// TIA Portal project "teste2" (V18)

(* hardware
DEVICE "S7-1200 station_1"  S7-1200 Station
   slot 0: "Rack_0"  S7-1200 Rack  Rack  V1.0
   slot 1: "PLC_1"  CPU 1214C AC/DC/Rly  6ES7 214-1BG40-0XB0  V4.5
   slot 2: "DI 16/DQ 16x24VDC_1"  6ES7 223-1BL32-0XB0  V2.0
   slot 3: "AI 8x13BIT_1"  6ES7 231-4HF32-0XB0  V2.1
*)

// ===== PLC "PLC_1"  CPU 1214C AC/DC/Rly =====

VAR_GLOBAL   // PLC tag table "Default tag table"
   "LED_Verde" AT %Q0.1 : Bool;
   "Bot_Emergencia" AT %I1.0 : Bool;
   "Bot_Verde" AT %I0.1 : Bool;
   "Tag_4" AT %M0.0 : Bool;
   "LED_Vermelho" AT %Q0.3 : Bool;
   "Bot_Reset" AT %I0.3 : Bool;
   "Parada" AT %M0.1 : Bool;
   "LED_Yellow" AT %Q0.2 : Bool;
   "Tag_1" AT %M0.2 : Bool;
   "Tag_2" AT %M0.3 : Bool;
   "Tag_3" AT %IW112 : Int;
   "norm" AT %MD68 : Real;
   "Angulo" AT %MW66 : Int;
   "Tag_5" AT %M0.6 : Bool;
END_VAR

TYPE "User_data_type_1"
   STRUCT
      Min_Norm : Int := 0;
      Max_Norm : Int := 27648;
   END_STRUCT;
END_TYPE

// folder: System blocks/Program resources

DATA_BLOCK "IEC_Timer_0_DB"   // DB1
{ S7_Optimized_Access := 'TRUE' }
AUTHOR : Simatic
FAMILY : IEC
NAME : IEC_TMR
VERSION : 1.0
// stored: InstanceOfName IEC_TIMER
"IEC_TIMER"
BEGIN
END_DATA_BLOCK

DATA_BLOCK "IEC_Timer_0_DB_1"   // DB2
{ S7_Optimized_Access := 'TRUE' }
AUTHOR : Simatic
FAMILY : IEC
NAME : IEC_TMR
VERSION : 1.0
// stored: InstanceOfName IEC_TIMER
"IEC_TIMER"
BEGIN
END_DATA_BLOCK

DATA_BLOCK "IEC_Timer_0_DB_2"   // DB3
{ S7_Optimized_Access := 'TRUE' }
AUTHOR : Simatic
FAMILY : IEC
NAME : IEC_TMR
VERSION : 1.0
// stored: InstanceOfName IEC_TIMER
"IEC_TIMER"
BEGIN
END_DATA_BLOCK

// folder: (top level)

ORGANIZATION_BLOCK "Main"   // OB1, LAD, ProgramCycle
TITLE = "Main Program Sweep (Cycle)"
{ S7_Optimized_Access := 'TRUE' }
VERSION : 0.1
   VAR_INPUT
      Initial_Call : Bool;   // Initial call of this OB
      Remanence : Bool;   // =True, if remanent data are available
   END_VAR
   VAR_TEMP   // added for the SCL form of the ladder/FBD networks
      _w1 : Bool;
      _w2 : Bool;
   END_VAR
BEGIN

REGION Network 1
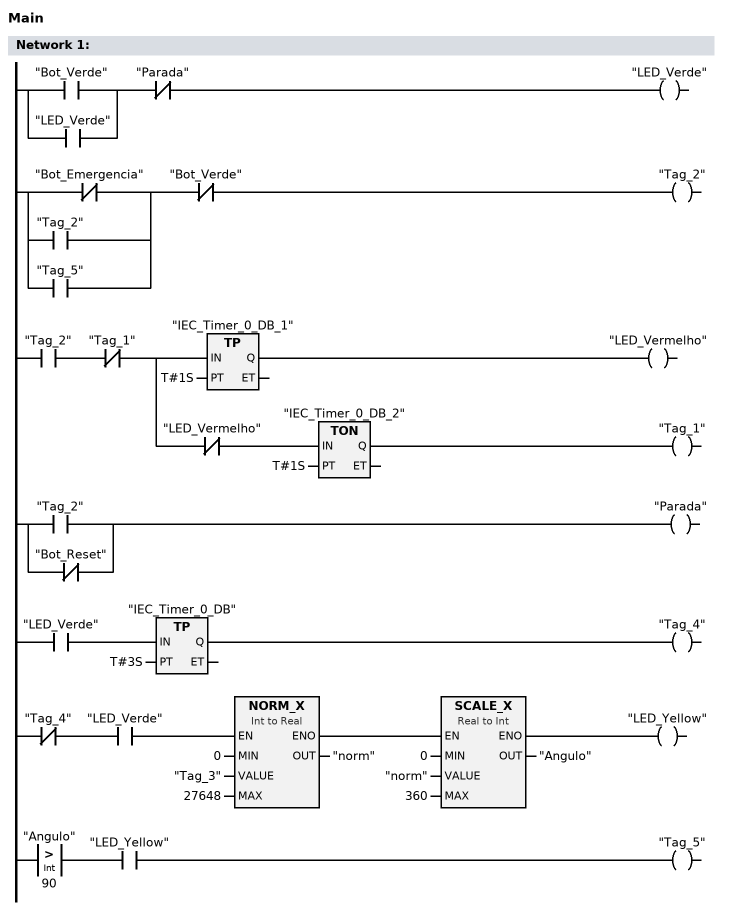
   "LED_Verde" := ("Bot_Verde" OR "LED_Verde") AND NOT "Parada";
   "Tag_2" := (NOT "Bot_Emergencia" OR "Tag_2" OR "Tag_5") AND NOT "Bot_Verde";
   #_w1 := "Tag_2" AND NOT "Tag_1";
   "IEC_Timer_0_DB_1".TP(IN := #_w1, PT := T#1S);
   "LED_Vermelho" := "IEC_Timer_0_DB_1".Q;
   "IEC_Timer_0_DB_2".TON(IN := #_w1 AND NOT "LED_Vermelho", PT := T#1S);
   "Tag_1" := "IEC_Timer_0_DB_2".Q;
   "Parada" := "Tag_2" OR NOT "Bot_Reset";
   "IEC_Timer_0_DB".TP(IN := "LED_Verde", PT := T#3S);
   "Tag_4" := "IEC_Timer_0_DB".Q;
   #_w2 := NOT "Tag_4" AND "LED_Verde";
   IF #_w2 THEN
       "norm" := NORM_X(MIN := 0, VALUE := "Tag_3", MAX := 27648);
       "Angulo" := SCALE_X(MIN := 0, VALUE := "norm", MAX := 360);
   END_IF;
   "LED_Yellow" := #_w2;
   "Tag_5" := ("Angulo" > 90) AND "LED_Yellow";
END_REGION
END_ORGANIZATION_BLOCK